Universal Robots PolyScope program: unalign_for_cover.urp

Program unalign_for_cover (installation=default directory=/programs createdIn=5.21.3 lastSavedIn=5.21.3 robotSerialNumber=20246801938)
Calibrated DH parameters: a=[-0.000071, -0.790281, -0.600694, 0.000061, -0.000039, 0]; d=[0.236272, 604.465945, 132.116513, -736.382239, 0.159268, 0.154005]; alpha=[1.570254, -0.000567, 0.000559, 1.571709, -1.56999, 0]; deltaTheta=[0, -0.409357, 7.293326, -0.600784, -0.000001, -0.000001]
InitVariablesNode
Robot Program (runOnlyOnce=true)
  SuppressedNode
    Folder dummypoints
      MoveJ speed 60 deg/s, acceleration 80 deg/s^2 (useActiveTCP=true optimoveEnabled=false optiMoveSpeed=0.3 optiMoveAcceleration=0.09) feature=Base
        'startpoint: oldhome'
        Waypoint Waypoint_1: TCP in base x=397.38 y=356.254 z=319.821 mm, rx=2.3163 ry=2.0576 rz=0.0741 rad; joints [-198.308, -118.162, 133.451, -12.562, -11.515, -6.325] deg; TCP offset x=-9.5 y=-328 z=105.73 mm, rx=1.2092 ry=-1.2092 rz=1.2092 rad
        'dummy left start'
        Waypoint Waypoint_2: TCP in base x=-1302.623 y=243.502 z=15.13 mm, rx=-2.912 ry=-1.1752 rz=-0.0069 rad; joints [-174.97, -153.223, -36.525, -170.672, 51.061, 0.264] deg
        'approach point near shoulder'
        Waypoint Waypoint_3: TCP in base x=-612.562 y=243.502 z=102.41 mm, rx=-2.912 ry=-1.1752 rz=-0.0069 rad; joints [-170.617, -105.873, -115.003, -139.508, 55.454, 0.207] deg
  SuppressedNode
    Folder actualprogram
      Folder liftcolumnup
        liftcolumnz := liftcolumnzneeded
        URCap MachineLogic for Universal Robots (MachineLogic for Universal Robots, Vention Inc.) dataModel(type=addMotor, numberAdded=0, speed_in_mm_per_min=600, acceleration_in_mm_per_s2=50.0, ActuatorPos=liftcolumnz, teachColor=BLUE, combo1=MachineMotion1, combo2=(1) Custom Actuator, combo3=Move to Position, combo6=In series, message=Move to Position, description=Moves the actuator to a specified position from the home location., comboAddress=Address 1, comboActuator=Valve 1)
      MoveJ speed 60 deg/s, acceleration 80 deg/s^2 (useActiveTCP=true optimoveEnabled=false optiMoveSpeed=0.3 optiMoveAcceleration=0.09) feature=Base
        Waypoint Waypoint_4: TCP in base x=-634.693 y=247.571 z=474.892 mm, rx=-2.4091 ry=-1.1113 rz=1.1282 rad; joints [-167.213, -64.784, -120.113, -130.92, 51.343, 6.187] deg
        Waypoint Waypoint_3: TCP in base x=-612.562 y=243.502 z=102.41 mm, rx=-2.912 ry=-1.1752 rz=-0.0069 rad; joints [-170.617, -105.873, -115.003, -139.508, 55.454, 0.207] deg
  SuppressedNode
    MoveJ speed 60 deg/s, acceleration 80 deg/s^2 (useActiveTCP=true optimoveEnabled=false optiMoveSpeed=0.3 optiMoveAcceleration=0.09) feature=Base
      'dummy points'
      Waypoint Waypoint_5: TCP in base x=-1008.914 y=279.358 z=44.412 mm, rx=-1.4579 ry=-0.6519 rz=0.6315 rad; joints [-159.825, -134.345, -108.311, -118.549, 63.05, 91.079] deg
      Waypoint Waypoint_6: TCP in base x=-1098.839 y=328.86 z=-127 mm, rx=-1.632 ry=-0.7226 rz=0.6064 rad; joints [-164.508, -143.465, -99.847, -116.758, -302.251, 80.059] deg
  SuppressedNode
    MoveJ speed 60 deg/s, acceleration 80 deg/s^2 (useActiveTCP=true optimoveEnabled=false optiMoveSpeed=0.3 optiMoveAcceleration=0.09) feature=Base
      Waypoint Waypoint_7: TCP in base x=-954.263 y=328.86 z=-127 mm, rx=-1.632 ry=-0.7226 rz=0.6064 rad; joints [-161.984, -139.644, -113.146, -107.279, -299.72, 80.058] deg
      Waypoint Waypoint_8: TCP in base x=-954.263 y=328.86 z=325.759 mm, rx=-1.632 ry=-0.7226 rz=0.6064 rad; joints [-161.997, -112.263, -109.215, -138.583, -299.736, 80.041] deg
  Folder actualprogram
    MoveL speed 250 mm/s, acceleration 1200 mm/s^2 (useActiveTCP=true optimoveEnabled=false optiMoveSpeed=0.3 optiMoveAcceleration=0.09) feature=Base
      MoveDirectionNode (selectedDirection=XPlus)
        Until DISTANCE (allowActions=false deceleration=3 distanceNodeType=STOP) Distance=0.15; motionParameters(blendRadius=0)
    MoveL speed 250 mm/s, acceleration 1200 mm/s^2 (useActiveTCP=true optimoveEnabled=false optiMoveSpeed=0.3 optiMoveAcceleration=0.09) feature=Base
      MoveDirectionNode (selectedDirection=ZPlus)
        Until DISTANCE (allowActions=false deceleration=3 distanceNodeType=STOP) Distance=0.2; motionParameters(blendRadius=0)
    MoveJ speed 60 deg/s, acceleration 80 deg/s^2 (useActiveTCP=true optimoveEnabled=false optiMoveSpeed=0.3 optiMoveAcceleration=0.09) feature=Base
      Waypoint Waypoint_9: TCP in base x=-242.109 y=328.86 z=325.759 mm, rx=-1.4053 ry=1.2267 rz=-1.0294 rad; joints [-207.989, -107.428, -116.696, -135.94, -215.722, 79.954] deg
      Waypoint Waypoint_10: TCP in base x=-240.92 y=326.607 z=327.046 mm, rx=-0.7835 ry=1.9486 rz=-1.6296 rad; joints [-234.825, -106.342, -118.044, -135.859, -188.602, 79.567] deg
    SafeHome (positionOptionType=SPEED_AND_ACCELERATION speed=1.047198 acceleration=1.396263 nextMotionTime=2)
    URCap MachineLogic for Universal Robots (MachineLogic for Universal Robots, Vention Inc.) dataModel(type=addMotor, numberAdded=0, combo1=MachineMotion1, combo2=(1) Custom Actuator, combo3=Home, combo6=In series, speed_in_mm_per_min=3000.0, acceleration_in_mm_per_s2=50.0, message=Homing, description=Moves the actuator in the negative direction until the home sensor is triggered and sets position to zero (0)., comboAddress=Address 1, comboActuator=Valve 1, teachColor=BLUE)
